PROGRAM p_Message
VAR_INPUT
  bReset        : BOOL;
  pListInternal : POINTER TO ARRAY[1..GVL_AXIS_CTRL.gciMaxMessage] OF ST_Message;
END_VAR
VAR_OUTPUT
  bActive       : BOOL;
  stMessageList : ST_MessageList;
END_VAR
VAR
  ui,uj,uk, ue  : INT := 1;
  bFoundEntry   : BOOL;
  iResetCount   : INT;
  atListWrite   : ARRAY[1..GVL_AXIS_CTRL.gciMaxMessage] OF ST_Message;
END_VAR


IF bReset
THEN
  bActive := FALSE;
  bReset  := FALSE;
  iResetCount := iResetCount + 1;
  stMessageList.sTextBox := '';

  memset(pListInternal, 0, SIZEOF(pListInternal^));
  memset(ADR(stMessageList.atMessages), 0, SIZEOF(stMessageList.atMessages));
  FOR uj :=  1 TO GVL_AXIS_CTRL.gciMaxMessage
  DO
    stMessageList.atMessages[uj].eType := '-1';
  END_FOR
END_IF

// copy to display list
FOR uk := ue TO GVL_AXIS_CTRL.gciMaxMessage
DO
  IF (pListInternal^[uk].udiError <> 0)
  THEN
    stMessageList.atMessages[uk].iErrorNumber := pListInternal^[uk].udiError;
    stMessageList.atMessages[uk].sTime        := pListInternal^[uk].tTime;
    stMessageList.atMessages[uk].sDevice      := DINT_TO_STRING(pListInternal^[uk].eDevice);
  ELSE
    EXIT;
  END_IF
END_FOR




// Look for text when message is selected
(*
(* Valid flag and iIndex coming from table visu element *)
IF stMessageList.bValid AND 
   stMessageList.iIndex <> stMessageList.iIndexOld
THEN
  stMessageList.sTextBox := '';

  IF pListInternal^[stMessageList.iIndex].eSubdevice >= e_SubDevice.SUB_DEVICE_AXIS_GENERAL
  THEN
    FOR ui := 1 TO cMaxMessagesNC
    DO
      IF GVL_NC_MESSAGES.gstNcAxisMessages[ui].id = stMessageList.atMessages[stMessageList.iIndex].iErrorNumber
      THEN
        stMessageList.sTextBox := GVL_NC_MESSAGES.gstNcAxisMessages[ui].FehlerText;
        EXIT;
      END_IF
    END_FOR
  (* TODO - append more Lists, e.g. ADS Errors *)
  END_IF
  stMessageList.iIndexOld := stMessageList.iIndex;
END_IF
*)

FOR uk := 1 TO GVL_AXIS_CTRL.gciMaxMessage
DO
  IF pListInternal^[uk].udiError <> 0
  THEN
    bActive := TRUE; // can be used for visual indication
  END_IF
END_FOR

END_PROGRAM

(* stored: Version 1.1.0.1, ProductVersion 3.1.4022.18
   POU p_Message: Id {73f25005-15f7-4639-abba-2bc02df878f8}, SpecialFunc None *)
